RoboDK station: Stringer B Corner-Bot-Short-BOX1.rdk

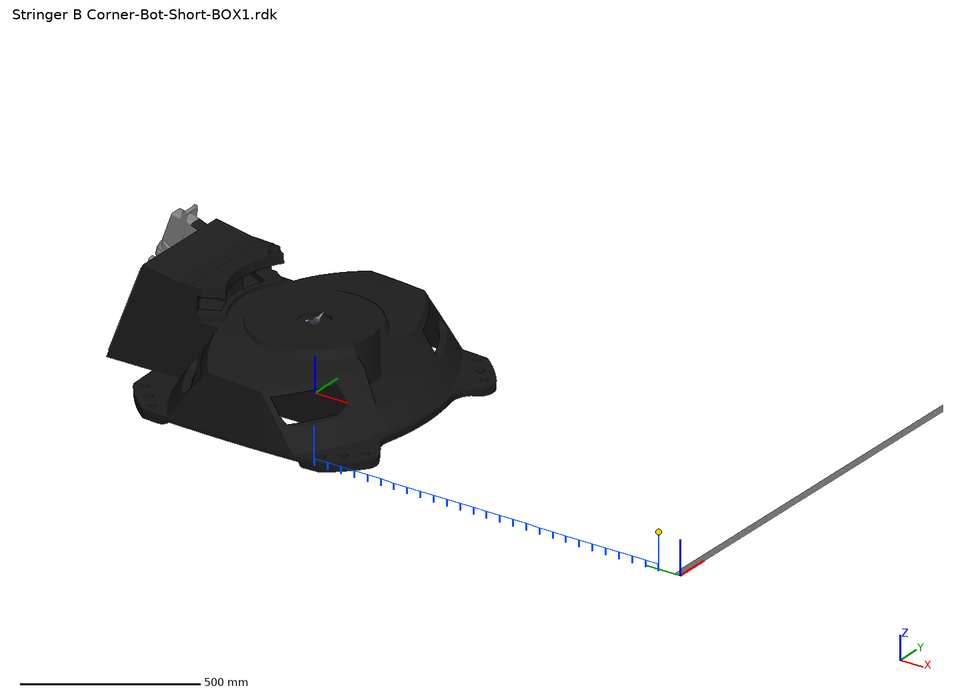
[picture v0: the station drawn from its stored meshes, robots at their saved joint values, targets as dots, program paths as lines]
Station Stringer B Corner-Bot-Short-BOX1 (saved by RoboDK 5.2.3). Poses are relative to the parent item; angles as X-Y-Z fixed-axis rotations.
  - frame KUKA KR 210 R2700 extra Base at (0, 0, 0) mm
    - robot KUKA KR 210 R2700 extra: 6 axes, payload 210 kg, reach 2696 mm, repeatability 0.06 mm, weight 1068 kg
        joint limits [-185, -140, -120, -350, -125, -350] to [185, -5, 155, 350, 125, 350]; home [0, -90, 90, 0, 0, 0]; saved at [-13.99, -56.961, 125.651, -207.973, 18.927, 195.716]
      - tool Spindle, TCP at (32, 0, 260) mm, rotated rx 0 ry 39 rz 0 deg, size 157.3 x 72 x 259.9 mm
  - frame Frame 2 at (1618.38, -541.41, 103.58) mm, rotated rx 0 ry 0 rz 90 deg
    - object L-Stringer B-bot-corner-short-BOX1 at (0, 0, 0) mm, size 1281.1 x 20 x 20 mm, geometry from L-Stringer B-bot-corner-short-BOX1.stl
    - object Stringer B Corner-Bot-Short-BOX1 at (0, 0, 0) mm, rotated rx 0 ry 0 rz -90 deg, 27 curves, geometry from Point 27
  - machining project Point settings: rotZ(0) | rotX(0)*rotY(0) | rotz(0) | onStart | onPathStart | onApproach | onPoint | onRetract | onFinish | SetRPM(%1) | SetTool(%1) | Extruder(%1) | default | default | OutOnMov(%1) | OutOffMov(%1) | onPathFinish | M_RunCode(%1)
  - machining project Point settings: rotZ(0) | rotX(0)*rotY(0) | rotz(0) | onStart | onPathStart | onApproach | onPoint | onRetract | onFinish | SetRPM(%1) | SetTool(%1) | Extruder(%1) | default | default | OutOnMov(%1) | OutOffMov(%1) | onPathFinish | M_RunCode(%1)
  - program Point (146 instructions, listed below)
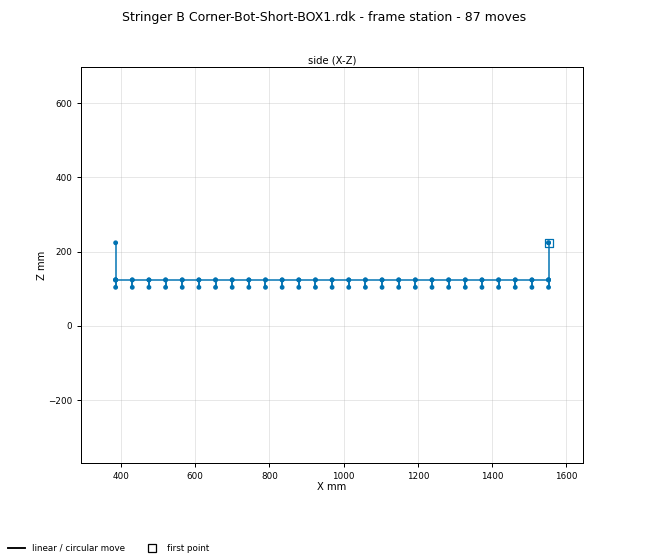
[picture p0: tool path of Stringer B Corner-Bot-Short-BOX1.rdk in frame station, 87 of 87 moves have a stored position in this frame; points joined in program order, loops and branches not executed]

--- program Point (robot KUKA KR 210 R2700 extra) ---
  Smooth(1)
  Set speed (1000.0 mm/s)
  Set Ref.: Frame 2
  Set Tool: Spindle
  Show Spindle
  MoveJ 1 to (-10.2, 66.57, 120) mm, rotated rx 180 ry 0 rz -180 deg; joints [19.592, -62.096, 124.056, -126.819, 15.284, 143.276]
  MoveL 2 to (-10.2, 66.57, 120) mm, rotated rx 180 ry 0 rz -180 deg; joints [19.592, -62.096, 124.056, -126.819, 15.284, 143.276]
  MoveL 3 to (-10.2, 66.57, 20) mm, rotated rx 180 ry 0 rz 180 deg; joints [19.592, -56.468, 123.483, -138.953, 18.745, 155.955]
  MoveL 4 to (-10.2, 66.57, 20) mm, rotated rx 180 ry 0 rz 180 deg; joints [19.592, -56.468, 123.483, -138.953, 18.745, 155.955]
  Set speed (50.0 mm/s)
  MoveL 5 to (-10.2, 66.57, 0) mm, rotated rx 180 ry 0 rz 180 deg; joints [19.592, -55.324, 123.308, -140.756, 19.485, 157.863]
  MoveL 6 to (-10.2, 66.57, 20) mm, rotated rx 180 ry 0 rz 180 deg; joints [19.592, -56.468, 123.483, -138.953, 18.745, 155.955]
  Set speed (1000.0 mm/s)
  MoveL 7 to (-10.2, 111.42, 20) mm, rotated rx -180 ry 0 rz -180 deg; joints [17.864, -56.782, 124.264, -142.945, 18.686, 158.488]
  Set speed (50.0 mm/s)
  MoveL 8 to (-10.2, 111.42, 0) mm, rotated rx -180 ry 0 rz -180 deg; joints [17.864, -55.623, 124.087, -144.622, 19.478, 160.262]
  MoveL 9 to (-10.2, 111.42, 20) mm, rotated rx -180 ry 0 rz -180 deg; joints [17.864, -56.782, 124.264, -142.945, 18.686, 158.488]
  Set speed (1000.0 mm/s)
  MoveL 10 to (-10.2, 156.26, 20) mm, rotated rx 180 ry 0 rz 180 deg; joints [16.103, -57.064, 124.971, -146.916, 18.649, 160.959]
  Set speed (50.0 mm/s)
  MoveL 11 to (-10.2, 156.26, 0) mm, rotated rx -180 ry 0 rz -180 deg; joints [16.103, -55.892, 124.793, -148.454, 19.49, 162.586]
  MoveL 12 to (-10.2, 156.26, 20) mm, rotated rx 180 ry 0 rz 180 deg; joints [16.103, -57.064, 124.971, -146.916, 18.649, 160.959]
  Set speed (1000.0 mm/s)
  MoveL 13 to (-10.2, 201.11, 20) mm, rotated rx -180 ry 0 rz -180 deg; joints [14.31, -57.316, 125.604, -150.864, 18.631, 163.369]
  Set speed (50.0 mm/s)
  MoveL 14 to (-10.2, 201.11, 0) mm, rotated rx 180 ry 0 rz -180 deg; joints [14.31, -56.13, 125.424, -152.249, 19.515, 164.835]
  MoveL 15 to (-10.2, 201.11, 20) mm, rotated rx -180 ry 0 rz -180 deg; joints [14.31, -57.316, 125.604, -150.864, 18.631, 163.369]
  Set speed (1000.0 mm/s)
  MoveL 16 to (-10.2, 245.96, 20) mm, rotated rx 180 ry 0 rz -180 deg; joints [12.487, -57.535, 126.162, -154.784, 18.626, 165.717]
  Set speed (50.0 mm/s)
  MoveL 17 to (-10.2, 245.96, 0) mm, rotated rx 180 ry 0 rz 180 deg; joints [12.487, -56.339, 125.981, -156.005, 19.549, 167.009]
  MoveL 18 to (-10.2, 245.96, 20) mm, rotated rx 180 ry 0 rz -180 deg; joints [12.487, -57.535, 126.162, -154.784, 18.626, 165.717]
  Set speed (1000.0 mm/s)
  MoveL 19 to (-10.2, 290.8, 20) mm, rotated rx 180 ry 0 rz 180 deg; joints [10.639, -57.724, 126.644, -158.673, 18.631, 168.003]
  Set speed (50.0 mm/s)
  MoveL 20 to (-10.2, 290.8, 0) mm, rotated rx -180 ry 0 rz -180 deg; joints [10.639, -56.517, 126.461, -159.723, 19.588, 169.114]
  MoveL 21 to (-10.2, 290.8, 20) mm, rotated rx 180 ry 0 rz 180 deg; joints [10.639, -57.724, 126.644, -158.673, 18.631, 168.003]
  Set speed (1000.0 mm/s)
  MoveL 22 to (-10.2, 335.65, 20) mm, rotated rx 180 ry 0 rz -180 deg; joints [8.768, -57.881, 127.048, -162.536, 18.641, 170.235]
  Set speed (50.0 mm/s)
  MoveL 23 to (-10.2, 335.65, 0) mm, rotated rx 180 ry 0 rz -180 deg; joints [8.768, -56.666, 126.864, -163.407, 19.628, 171.157]
  MoveL 24 to (-10.2, 335.65, 20) mm, rotated rx 180 ry 0 rz -180 deg; joints [8.768, -57.881, 127.048, -162.536, 18.641, 170.235]
  Set speed (1000.0 mm/s)
  MoveL 25 to (-10.2, 380.5, 20) mm, rotated rx -180 ry 0 rz -180 deg; joints [6.878, -58.008, 127.373, -166.373, 18.654, 172.419]
  Set speed (50.0 mm/s)
  MoveL 26 to (-10.2, 380.5, 0) mm, rotated rx 180 ry 0 rz -180 deg; joints [6.878, -56.785, 127.189, -167.059, 19.664, 173.145]
  MoveL 27 to (-10.2, 380.5, 20) mm, rotated rx -180 ry 0 rz -180 deg; joints [6.878, -58.008, 127.373, -166.373, 18.654, 172.419]
  Set speed (1000.0 mm/s)
  MoveL 28 to (-10.2, 425.34, 20) mm, rotated rx 180 ry 0 rz 180 deg; joints [4.972, -58.103, 127.62, -170.187, 18.666, 174.562]
  Set speed (50.0 mm/s)
  MoveL 29 to (-10.2, 425.34, 0) mm, rotated rx 180 ry 0 rz -180 deg; joints [4.972, -56.875, 127.435, -170.685, 19.695, 175.089]
  MoveL 30 to (-10.2, 425.34, 20) mm, rotated rx 180 ry 0 rz 180 deg; joints [4.972, -58.103, 127.62, -170.187, 18.666, 174.562]
  Set speed (1000.0 mm/s)
  MoveL 31 to (-10.2, 470.19, 20) mm, rotated rx -180 ry 0 rz -180 deg; joints [3.056, -58.167, 127.787, -173.986, 18.676, 176.676]
  Set speed (50.0 mm/s)
  MoveL 32 to (-10.2, 470.19, 0) mm, rotated rx -180 ry 0 rz -180 deg; joints [3.056, -56.936, 127.602, -174.293, 19.716, 177.001]
  MoveL 33 to (-10.2, 470.19, 20) mm, rotated rx -180 ry 0 rz -180 deg; joints [3.056, -58.167, 127.787, -173.986, 18.676, 176.676]
  Set speed (1000.0 mm/s)
  MoveL 34 to (-10.2, 515.03, 20) mm, rotated rx 180 ry 0 rz 180 deg; joints [1.133, -58.201, 127.874, -177.774, 18.681, 178.771]
  Set speed (50.0 mm/s)
  MoveL 35 to (-10.2, 515.03, 0) mm, rotated rx -180 ry 0 rz -180 deg; joints [1.133, -56.967, 127.689, -177.887, 19.728, 178.892]
  MoveL 36 to (-10.2, 515.03, 20) mm, rotated rx 180 ry 0 rz 180 deg; joints [1.133, -58.201, 127.874, -177.774, 18.681, 178.771]
  Set speed (1000.0 mm/s)
  MoveL 37 to (-10.2, 559.88, 20) mm, rotated rx 180 ry 0 rz 180 deg; joints [-0.793, -58.203, 127.882, -181.558, 18.682, 180.86]
  Set speed (50.0 mm/s)
  MoveL 38 to (-10.2, 559.88, 0) mm, rotated rx 180 ry 0 rz -180 deg; joints [-0.793, -56.97, 127.696, -181.478, 19.729, 180.775]
  MoveL 39 to (-10.2, 559.88, 20) mm, rotated rx 180 ry 0 rz 180 deg; joints [-0.793, -58.203, 127.882, -181.558, 18.682, 180.86]
  Set speed (1000.0 mm/s)
  MoveL 40 to (-10.2, 604.73, 20) mm, rotated rx 180 ry 0 rz 180 deg; joints [-2.717, -58.175, 127.808, -185.345, 18.677, 182.953]
  Set speed (50.0 mm/s)
  MoveL 41 to (-10.2, 604.73, 0) mm, rotated rx -180 ry 0 rz -180 deg; joints [-2.717, -56.943, 127.623, -185.073, 19.719, 182.664]
  MoveL 42 to (-10.2, 604.73, 20) mm, rotated rx 180 ry 0 rz 180 deg; joints [-2.717, -58.175, 127.808, -185.345, 18.677, 182.953]
  Set speed (1000.0 mm/s)
  MoveL 43 to (-10.2, 649.57, 20) mm, rotated rx -180 ry 0 rz -180 deg; joints [-4.635, -58.116, 127.655, -189.141, 18.668, 185.063]
  Set speed (50.0 mm/s)
  MoveL 44 to (-10.2, 649.57, 0) mm, rotated rx -180 ry 0 rz -180 deg; joints [-4.635, -56.888, 127.47, -188.677, 19.699, 184.571]
  MoveL 45 to (-10.2, 649.57, 20) mm, rotated rx -180 ry 0 rz -180 deg; joints [-4.635, -58.116, 127.655, -189.141, 18.668, 185.063]
  Set speed (1000.0 mm/s)
  MoveL 46 to (-10.2, 694.42, 20) mm, rotated rx 180 ry 0 rz 180 deg; joints [-6.542, -58.027, 127.423, -192.953, 18.656, 187.201]
  Set speed (50.0 mm/s)
  MoveL 47 to (-10.2, 694.42, 0) mm, rotated rx 180 ry 0 rz 180 deg; joints [-6.542, -56.803, 127.238, -192.3, 19.67, 186.509]
  MoveL 48 to (-10.2, 694.42, 20) mm, rotated rx 180 ry 0 rz 180 deg; joints [-6.542, -58.027, 127.423, -192.953, 18.656, 187.201]
  Set speed (1000.0 mm/s)
  MoveL 49 to (-10.2, 739.26, 20) mm, rotated rx -180 ry 0 rz -180 deg; joints [-8.435, -57.906, 127.111, -196.785, 18.643, 189.376]
  Set speed (50.0 mm/s)
  MoveL 50 to (-10.2, 739.26, 0) mm, rotated rx -180 ry 0 rz -180 deg; joints [-8.435, -56.689, 126.927, -195.946, 19.635, 188.488]
  MoveL 51 to (-10.2, 739.26, 20) mm, rotated rx -180 ry 0 rz -180 deg; joints [-8.435, -57.906, 127.111, -196.785, 18.643, 189.376]
  Set speed (1000.0 mm/s)
  MoveL 52 to (-10.2, 784.11, 20) mm, rotated rx 180 ry 0 rz -180 deg; joints [-10.31, -57.754, 126.721, -200.643, 18.632, 191.599]
  Set speed (50.0 mm/s)
  MoveL 53 to (-10.2, 784.11, 0) mm, rotated rx 180 ry 0 rz 180 deg; joints [-10.31, -56.545, 126.538, -199.624, 19.595, 190.521]
  MoveL 54 to (-10.2, 784.11, 20) mm, rotated rx 180 ry 0 rz -180 deg; joints [-10.31, -57.754, 126.721, -200.643, 18.632, 191.599]
  Set speed (1000.0 mm/s)
  MoveL 55 to (-10.2, 828.96, 20) mm, rotated rx -180 ry 0 rz -180 deg; joints [-12.163, -57.571, 126.253, -204.528, 18.626, 193.876]
  Set speed (50.0 mm/s)
  MoveL 56 to (-10.2, 828.96, 0) mm, rotated rx -180 ry 0 rz -180 deg; joints [-12.163, -56.372, 126.071, -203.336, 19.556, 192.614]
  MoveL 57 to (-10.2, 828.96, 20) mm, rotated rx -180 ry 0 rz -180 deg; joints [-12.163, -57.571, 126.253, -204.528, 18.626, 193.876]
  Set speed (1000.0 mm/s)
  MoveL 58 to (-10.2, 873.8, 20) mm, rotated rx 180 ry 0 rz 180 deg; joints [-13.99, -57.357, 125.708, -208.442, 18.629, 196.212]
  Set speed (50.0 mm/s)
  MoveL 59 to (-10.2, 873.8, 0) mm, rotated rx 180 ry 0 rz 180 deg; joints [-13.99, -56.169, 125.528, -207.085, 19.521, 194.776]
  MoveL 60 to (-10.2, 873.8, 20) mm, rotated rx 180 ry 0 rz 180 deg; joints [-13.99, -57.357, 125.708, -208.442, 18.629, 196.212]
  Set speed (1000.0 mm/s)
  MoveL 61 to (-10.2, 918.65, 20) mm, rotated rx -180 ry 0 rz -180 deg; joints [-15.789, -57.111, 125.088, -212.385, 18.645, 198.61]
  Set speed (50.0 mm/s)
  MoveL 62 to (-10.2, 918.65, 0) mm, rotated rx 180 ry 0 rz -180 deg; joints [-15.789, -55.936, 124.91, -210.873, 19.493, 197.011]
  MoveL 63 to (-10.2, 918.65, 20) mm, rotated rx -180 ry 0 rz -180 deg; joints [-15.789, -57.111, 125.088, -212.385, 18.645, 198.61]
  Set speed (1000.0 mm/s)
  MoveL 64 to (-10.2, 963.5, 20) mm, rotated rx 180 ry 0 rz -180 deg; joints [-17.556, -56.834, 124.394, -216.353, 18.678, 201.072]
  Set speed (50.0 mm/s)
  MoveL 65 to (-10.2, 963.5, 0) mm, rotated rx 180 ry 0 rz -180 deg; joints [-17.556, -55.673, 124.217, -214.699, 19.479, 199.322]
  MoveL 66 to (-10.2, 963.5, 20) mm, rotated rx 180 ry 0 rz -180 deg; joints [-17.556, -56.834, 124.394, -216.353, 18.678, 201.072]
  Set speed (1000.0 mm/s)
  MoveL 67 to (-10.2, 1008.34, 20) mm, rotated rx 180 ry 0 rz 180 deg; joints [-19.289, -56.525, 123.626, -220.341, 18.732, 203.594]
  Set speed (50.0 mm/s)
  MoveL 68 to (-10.2, 1008.34, 0) mm, rotated rx 180 ry 0 rz -180 deg; joints [-19.289, -55.379, 123.451, -218.559, 19.483, 201.708]
  MoveL 69 to (-10.2, 1008.34, 20) mm, rotated rx 180 ry 0 rz 180 deg; joints [-19.289, -56.525, 123.626, -220.341, 18.732, 203.594]
  Set speed (1000.0 mm/s)
  MoveL 70 to (-10.2, 1053.19, 20) mm, rotated rx 180 ry 0 rz -180 deg; joints [-20.987, -56.185, 122.787, -224.343, 18.813, 206.172]
  Set speed (50.0 mm/s)
  MoveL 71 to (-10.2, 1053.19, 0) mm, rotated rx 180 ry 0 rz 180 deg; joints [-20.987, -55.054, 122.613, -222.449, 19.509, 204.167]
  MoveL 72 to (-10.2, 1053.19, 20) mm, rotated rx 180 ry 0 rz -180 deg; joints [-20.987, -56.185, 122.787, -224.343, 18.813, 206.172]
  Set speed (1000.0 mm/s)
  MoveL 73 to (-10.2, 1098.03, 20) mm, rotated rx -180 ry 0 rz -180 deg; joints [-22.647, -55.813, 121.876, -228.348, 18.923, 208.798]
  Set speed (50.0 mm/s)
  MoveL 74 to (-10.2, 1098.03, 0) mm, rotated rx 180 ry 0 rz -180 deg; joints [-22.647, -54.698, 121.705, -226.361, 19.562, 206.693]
  MoveL 75 to (-10.2, 1098.03, 20) mm, rotated rx -180 ry 0 rz -180 deg; joints [-22.647, -55.813, 121.876, -228.348, 18.923, 208.798]
  Set speed (1000.0 mm/s)
  MoveL 76 to (-10.2, 1142.88, 20) mm, rotated rx 180 ry 0 rz 180 deg; joints [-24.267, -55.41, 120.897, -232.347, 19.068, 211.465]
  Set speed (50.0 mm/s)
  MoveL 77 to (-10.2, 1142.88, 0) mm, rotated rx -180 ry 0 rz -180 deg; joints [-24.267, -54.312, 120.727, -230.285, 19.648, 209.279]
  MoveL 78 to (-10.2, 1142.88, 20) mm, rotated rx 180 ry 0 rz 180 deg; joints [-24.267, -55.41, 120.897, -232.347, 19.068, 211.465]
  Set speed (1000.0 mm/s)
  MoveL 79 to (-10.2, 1187.73, 20) mm, rotated rx 180 ry 0 rz 180 deg; joints [-25.848, -54.975, 119.849, -236.327, 19.25, 214.159]
  Set speed (50.0 mm/s)
  MoveL 80 to (-10.2, 1187.73, 0) mm, rotated rx 180 ry 0 rz 180 deg; joints [-25.848, -53.894, 119.681, -234.21, 19.77, 211.913]
  MoveL 81 to (-10.2, 1187.73, 20) mm, rotated rx 180 ry 0 rz 180 deg; joints [-25.848, -54.975, 119.849, -236.327, 19.25, 214.159]
  Set speed (1000.0 mm/s)
  MoveL 82 to (-10.2, 1232.57, 20) mm, rotated rx -180 ry 0 rz -180 deg; joints [-27.387, -54.508, 118.735, -240.274, 19.472, 216.869]
  Set speed (50.0 mm/s)
  MoveL 83 to (-10.2, 1232.57, 0) mm, rotated rx -180 ry 0 rz 180 deg; joints [-27.387, -53.445, 118.569, -238.122, 19.932, 214.584]
  MoveL 84 to (-10.2, 1232.57, 20) mm, rotated rx -180 ry 0 rz -180 deg; joints [-27.387, -54.508, 118.735, -240.274, 19.472, 216.869]
  MoveL 85 to (-10.2, 1232.57, 20) mm, rotated rx -180 ry 0 rz -180 deg; joints [-27.387, -54.508, 118.735, -240.274, 19.472, 216.869]
  Set speed (1000.0 mm/s)
  MoveL 86 to (-10.2, 1232.57, 20) mm, rotated rx -180 ry 0 rz -180 deg; joints [-27.387, -54.508, 118.735, -240.274, 19.472, 216.869]
  MoveL 87 to (-10.2, 1232.57, 120) mm, rotated rx -180 ry 0 rz -180 deg; joints [-27.387, -59.725, 119.278, -253.107, 17.61, 230.397]
